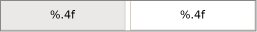
VISUALIZATION VISU_ConfigLREAL4Entry  // 257x32
VAR_IN_OUT
    active : LREAL;
    editable : LREAL;
END_VAR
    Textfield (0,0 125x30), "%.4f", text variable: active, input disabled if: TRUE
    Textfield (130,0 125x30), "%.4f", text variable: editable, colour toggle: editable <> active
        OnMouseClick: write the text variable via Default
END_VISUALIZATION

(* stored: Version 1.1.0.1, ProductVersion 3.1.0.36
   Visu VISU_ConfigLREAL4Entry: Id {eeef9d02-ed3f-467e-8aff-83760e7cb3f5} *)
